% RSLogix 500 project I2P Job 07 - Leo Kniffen.RSS, saved by version 10.00.00.00 %
PROJECT "ML04B"    % processor: Bul.1763 MicroLogix 1100 Series B %

PROGRAM FILES
  LAD 2   3 rungs

DATA FILES
  O0 OUTPUT  4 elements
  I1 INPUT  6 elements
  S2 STATUS  66 elements
  B3 BINARY  1 elements
  T4 TIMER  1 elements
  C5 COUNTER  1 elements
  R6 CONTROL  1 elements
  N7 INTEGER  1 elements
  F8 FLOAT  1 elements

LADDER 2
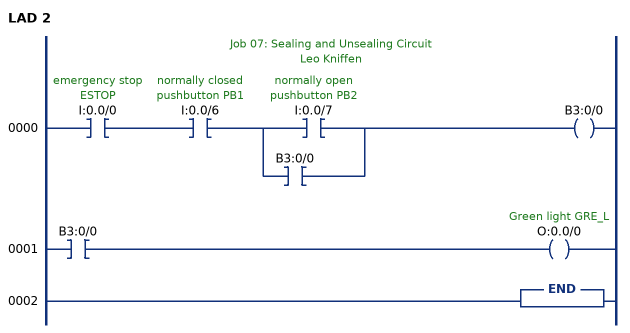
% Rung: 0 %
% Job 07: Sealing and Unsealing Circuit
% Leo Kniffen %
SOR XIC I:0.0/0 XIC I:0.0/6 BST XIC I:0.0/7 NXB XIC B3:0/0 BND OTE B3:0/0 EOR
%   I:0.0/0  ESTOP  "emergency stop" %
%   I:0.0/6  PB1  "normally closed pushbutton" %
%   I:0.0/7  PB2  "normally open pushbutton" %
% Rung: 1 %
SOR XIC B3:0/0 OTE O:0.0/0 EOR
%   O:0.0/0  GRE_L  "Green light" %
% Rung: 2 %
SOR END EOR

OTHER DOCUMENTED ADDRESSES
  I:0.0/1  CR1_CON  "control relay 1 contacts"
  I:0.0/2  CR2_CON  "control relay 2 contacts"
  I:0.0/3  3PSS_A  "3 position selector switch position A"
  I:0.0/4  3PSS_B  "3 position selector switch position B"
  I:0.0/5  2PSS  "2 position selector switch"
  I:0.0/8  PB3  "normally open pushbutton"
  O:0.0/1  YEL_L  "yellow light"
  O:0.0/2  RED_L  "red light"
  O:0.0/3  BLU_L  "blue light"
  O:0.0/4  CR1  "control relay 1-8 pin"
  O:0.0/5  CR2  "control relay 2-11 pin"
